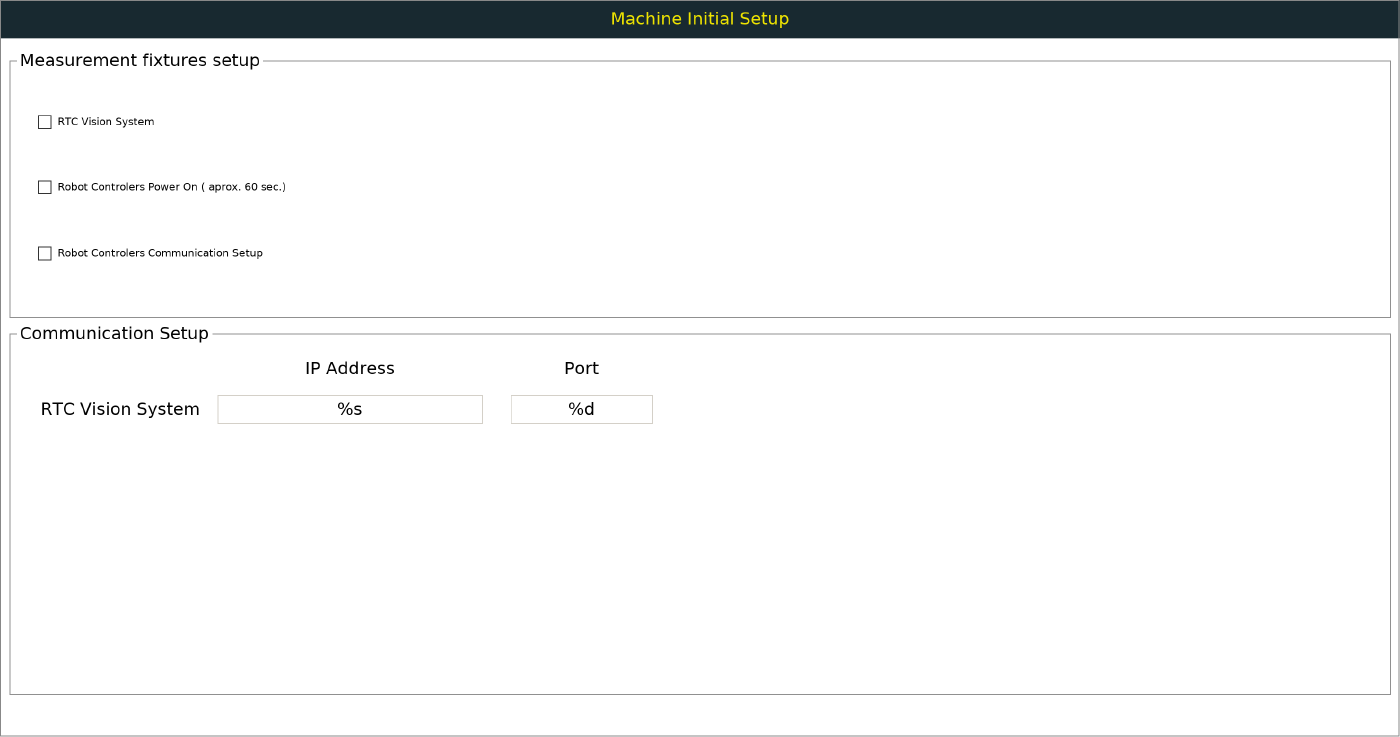
VISUALIZATION UninitializedSetupFrame  // 1480x780
VAR_IN_OUT
	//stUninitializedFrame : ST_UninitializedSetupFrame;
END_VAR
    GroupBox (10,56 1460x280), "Measurement fixtures setup"
        Checkbox (28,58 400x30), "RTC Vision System"
        Checkbox (28,127 450x30), "Robot Controlers Power On ( aprox. 60 sec.)"
        Checkbox (28,197 400x30), "Robot Controlers Communication Setup"
    GroupBox (10,345 1460x390), "Communication Setup"
        Label (30,63 192x50), "RTC Vision System"
        Textfield (220,73 280x30), "%s"
            OnMouseClick: write the text variable via VisuDialogs.Numpad
        Textfield (530,73 150x30), "%d"
            OnMouseClick: write the text variable via VisuDialogs.Numpad
        Label (220,30 280x30), "IP Address"
        Label (530,30 150x30), "Port"
    Rectangle (0,0 1480x40), "Machine Initial Setup"
END_VISUALIZATION

(* stored: Version 1.1.0.1, ProductVersion 3.1.4024.9
   Visu UninitializedSetupFrame: Id {e3d78ec9-da04-4d79-9198-ce14237d1d82} *)
